# B&R Automation Studio project Lab4
Automation Studio 4.5.2.102

## Logical view

Binary libraries used (declarations not repeated): Runtime, Operator, AsIecCon, astime, sys_lib, asstring, Acp10man, Acp10par, NcGlobal, Acp10sdc, Acp10_MC, brsystem, AsBrStr, Acp10sim, AsIOTime, MotrContr

### Global.var - Global variables
```iecst
VAR
	gAxis_X : ACP10AXIS_typ := (0);
	gAxis_X_HW : SdcHwCfg_typ := (0);
	gAxis_X_DrvIf : SdcDrvIf16_typ := (0);
	gAxis_X_DiDoIf : SdcDiDoIf_typ := (0);
	gAxis_X_EncIf : SdcEncIf16_typ := (0);
END_VAR
```


Listed in the project but not available here: Logical/Global.typ, Logical/acp10etxen, Logical/gAxis_X, Logical/SDCAxisCtrlX
